// Mitsubishi GX Works2 project: ventilationUnitStart_exp   PLC: FX3G
// Базовая структура управления вентиляциооной установкой

// global labels: Global1
VAR_GLOBAL
  xStart AT M10 : BOOL;  (* Переменная разрешения на работу установки *)
  xSeason AT M12 : BOOL;  (* Определение сезона 0 - Зима 1 - Лето *)
  xAlarm AT M1 : BOOL;  (* Общий статус Аварий 0 - нет 1 - Авария *)
  xWarning AT M2 : BOOL;  (* Общий статус предупреждений 0 - нет 1 - есть предупреждения *)
  dI_AlarmFreeze AT X000 : BOOL;  (* Авария термостата заморозки *)
  xAlarmSensors AT M7 : BOOL;  (* Общая аврия Датчиков - всне диапазона *)
  dI_AlarmPumpWater AT X001 : BOOL;  (* Авария насоса (сработка защиты) *)
  dI_AlarmMotorSupply AT X002 : BOOL;  (* Авария реле Вентилятора Притока *)
  dI_AlarmMotorExhaust AT X003 : BOOL;  (* Авария реле Вентилятора Вытяжки *)
  dI_WarnPresFilterSupply AT X007 : BOOL;  (* Авария пресостата фильтра Притока *)
  dI_WarnPresFilterExaust AT X006 : BOOL;  (* Авария пресостата фильтра Вытяжки *)
  dI_AlarmPresMotorSupply AT X004 : BOOL;  (* Авария пресостата вентилятора Притока *)
  dI_AlarmPresMotorExhaust AT X005 : BOOL;  (* Авария пресостата вентилятора Вытяжки *)
  xAlarmWarmWater AT M8 : BOOL;  (* Авария снижения температуры теплоносителя темплообменника - Требуется прогрев *)
  wDeltaTempOut AT D11 : INT;  (* Значение смещения показаний датчика (корректировка) *)
  wDeltaTempInRoom AT D10 : INT;  (* Значение смещения показаний датчика (корректировка) *)
  wDeltaTempFromRoom AT D9 : INT;  (* Значение смещения показаний датчика (корректировка) *)
  wDeltaTempEmpty AT D8 : INT;  (* Значение смещения показаний датчика (корректировка) *)
  xAlarmSensorOut AT M6 : BOOL;  (* Авария датчика Наружней температуры *)
  xAlarmSensorInRoom AT M5 : BOOL;  (* Авария датчика температуры Подачи В помещение *)
  xAlarmSensorFromRoom AT M4 : BOOL;  (* Авария датчика температуры забираемого ИЗ помещения *)
  xAlarmSensorEmpty AT M3 : BOOL;  (* Авария датчика температуры *)
  iR_TempOut AT D6 : WORD;  (* Значение сопротивление линии связи резистивного датчика *)
  iR_TempInRoom AT D5 : WORD;  (* Значение сопротивление линии связи резистивного датчика *)
  iR_TempFromRoom AT D4 : WORD;  (* Значение сопротивление линии связи резистивного датчика *)
  iRTempEmpty AT D7 : WORD;  (* Значение сопротивление линии связи резистивного датчика *)
  dO_PumpStart AT Y004 : BOOL;  (* Разрешение на работу Насоса контура водяного теплообменника *)
  dO_SupplyMotorStart AT Y003 : BOOL;  (* Разрешение на запуск Вентилятора Притока *)
  dO_ExhaustMotorStart AT Y001 : BOOL;  (* Разрешение на запуск Вентилятора Вытяжки *)
  dO_SupplyDamperStart AT Y002 : BOOL;  (* Разрешение на открытие Заслонки Притока *)
  dO_ExhaustDamperStart AT Y000 : BOOL;  (* Разрешение на открытие Заслонки Вытяжки *)
  iDelayStart AT D2 : WORD;  (* Значение задержки (общее) *)
  iDelaySupplyMotor AT D3 : WORD;  (* Значение задержки пуска Вентилятора Притока *)
  iDelayExhaustMotor AT D1 : WORD;  (* Значение задержки пуска Вентилятора Вытяжки *)
  iDelayDamper AT D0 : WORD;  (* Значение задержки открытия заслонки *)
  xUserStart AT M11 : BOOL;  (* Переменная изменяемая Пользователем для разрешения работы *)
  xUserSeason AT M13 : BOOL;  (* Переменная изменяемая Пользователем для выбора Сезона *)
  xUserArarmReset AT M14 : BOOL;  (* Переменная изменяемая Пользователем для сброса общего флага Аварий *)
  xAlarmCritical AT M0 : BOOL;  (* Cтатус критических Аварий 0 - нет 1 - Авария *)
  xInit AT M15 : BOOL;  (* Переменная разрешающая иницилизацию при старте *)
  aI_TempOut AT D14 : INT;  (* AI_0 Датчик наружней температуры D8030 *)
  aI_TempSupply AT D15 : INT;  (* AI_1 Датчик притока (температуры подачи в помещение)  D8031 *)
  aI_TempWater AT D16 : INT;  (* AI_2 Датчик обратной воды  D8032 *)
  aI_TempRecupOut AT D17 : INT;  (* AI_3 Датчик температуры за рекуператором  D8033 *)
  aO_1 AT D8050 : REAL;  (* AO_ Первый аналоговый D8050 *)
  aO_2 AT D8051 : REAL;  (* AO_ Второй аналоговый выход D8051 *)
  iUserTempSummer AT D12 : INT;  (* Температура перехода на летний режим *)
  iUserTemWinter AT D13 : INT;  (* Температура перехода на зимний режим *)
  aI_TempFromRoom AT D18 : INT;  (* AI_4 Датчик вытяжной температуры из помещения D8034 *)
  iUserAccess AT D40 : WORD;  (* Уровень доступа текущего пользователя *)
  iUserSetpoint AT D20 : INT;  (* Уставка *)
  testTempOut AT D41 : INT;  (* Тестирование перехода   Зима/Лето *)
END_VAR

// task Task_01 (event TRUE, interval 0, priority 31): POU_01
// task Init (event TRUE, interval 0, priority 1): Init
// user libraries (not included): AlarmManger128, Utils

PROGRAM Init
VAR
  fbAmSet : AM_SET;
  fbAmInit : AM_INIT;
  fbAmIs : AM_HAS_ALARMS;
  fbAmBlockIs : AM_IS_BLOCK;
  fbAmEvents : AM_EVENT;
  fbAmRST : AM_RST;
  fbAmEventRST : AM_EVENT_RESET;
END_VAR
(*Programm is run only one time when plc started to initiate alarms,  warnings and configuration settings *)

(* Init PID*)

(*Init Alarms *)
IF NOT xInit THEN 
	AM_D_START :=3000; (* Start alarms library*)
	
	(* Critical Alarm signals*)
	 fbAmInit(iNum := 0, iSeverity :=4, iProcess :=1, xLock := TRUE, xLatch := TRUE,  xBuzzer := TRUE ); (*Fire alarm *)
	 fbAmInit(iNum := 1, iSeverity :=4, iProcess :=1, xLock := TRUE, xLatch := TRUE,  xBuzzer := TRUE ); (*Freeze alarm *)
	 fbAmInit(iNum := 2, iSeverity :=4, iProcess :=1, xLock := TRUE, xLatch := TRUE,  xBuzzer := TRUE ); (*Warming Up the water circuit*)
	 fbAmInit(iNum := 4, iSeverity :=4, iProcess :=1, xLock := TRUE, xLatch := TRUE,  xBuzzer := TRUE ); (*Critical alarm the water circuit*)
	  
	 (* Air Presure sensors*)
	 fbAmInit(iNum := 5, iSeverity :=2, iProcess :=2, xLock := TRUE, xLatch := FALSE,  xBuzzer := TRUE ); (*Supply filter *)
	 fbAmInit(iNum := 6, iSeverity :=2, iProcess :=2, xLock := TRUE, xLatch := FALSE,  xBuzzer := TRUE ); (*Exhaust filter *)
	 fbAmInit(iNum := 7, iSeverity :=3, iProcess :=2, xLock := TRUE, xLatch := FALSE,  xBuzzer := TRUE ); (*Supply motor air alarm *)
	 fbAmInit(iNum := 8, iSeverity :=3, iProcess :=2, xLock := TRUE, xLatch := FALSE,  xBuzzer := TRUE ); (*Exhaust motor air alarm *)
	 (* Vent Motors Alarm sensors*)
	 fbAmInit(iNum := 9, iSeverity :=3, iProcess :=3, xLock := TRUE, xLatch := FALSE,  xBuzzer := TRUE ); (*Supply motor Alarm *)
	 fbAmInit(iNum := 10, iSeverity :=3, iProcess :=3, xLock := TRUE, xLatch := FALSE,  xBuzzer := TRUE ); (*Exhaust motor Alarm *)
	 (* Pumpsr Alarm sensors*)
	 fbAmInit(iNum := 11, iSeverity :=3, iProcess :=3, xLock := TRUE, xLatch := FALSE,  xBuzzer := TRUE ); (*Pump water Alarm*)
	 fbAmInit(iNum := 12, iSeverity :=3, iProcess :=3, xLock := TRUE, xLatch := FALSE,  xBuzzer := TRUE ); (*Pump glycol Alarm*)
	 (* Temperature sensors*)
	 fbAmInit(iNum := 13, iSeverity :=2, iProcess :=4, xLock := TRUE, xLatch := FALSE,  xBuzzer := TRUE ); (*Temp out *)
	 fbAmInit(iNum := 14,  iSeverity :=2, iProcess :=4, xLock := TRUE, xLatch := FALSE,  xBuzzer := TRUE ); (*Temp supply in room *)
	 fbAmInit(iNum := 15,  iSeverity :=2, iProcess :=4, xLock := TRUE, xLatch := FALSE,  xBuzzer := TRUE ); (*Temp exhaust from room *)
	 fbAmInit(iNum := 16,  iSeverity :=2, iProcess :=4, xLock := TRUE, xLatch := FALSE,  xBuzzer := TRUE ); (*Temp after recuperation *)
	 fbAmInit(iNum := 17,  iSeverity :=2, iProcess :=4, xLock := TRUE, xLatch := FALSE,  xBuzzer := TRUE ); (*Temp water return *)
	 fbAmInit(iNum := 18,  iSeverity :=2, iProcess :=4, xLock := TRUE, xLatch := FALSE,  xBuzzer := TRUE ); (*Temp glycol return *)
	 
	 (* SeasonControl*)
	 fbAmInit(iNum := 30,  iSeverity :=1, iProcess :=5, xLock := FALSE, xLatch := FALSE,  xBuzzer := FALSE); (*start Winter Season *)
	 fbAmInit(iNum := 31,  iSeverity :=1, iProcess :=5, xLock := FALSE, xLatch := FALSE,  xBuzzer := FALSE); (*start SammerSeason *)
	 
	 (* Init ModBus*)
	 
	 
	 
	xInit := TRUE;	
END_IF ;

(* *)
END_PROGRAM

PROGRAM POU_01
VAR
  iStep : INT;
  fbAmSet : AM_SET;
  fbAmInit : AM_INIT;
  fbAmIs : AM_HAS_ALARMS;
  fbAmBlockIs : AM_IS_BLOCK;
  fbAmEvents : AM_EVENT;
  fbAmRST : AM_RST;
  fbAmEventRST : AM_EVENT_RESET;
  localSeasonTriger : BOOL;
  icountMin : INT;
  init : INT;
END_VAR
(* RST( MEP( xManualWorks ) , xAutoWorks );
RST( MEP(xAutoWorks ) ,xManualWorks  );  *)
(* System can work only in one state Auto or Manual There is constol change*)

(* IF iStep <> 10 THEN iStep := 0; END_IF; *)

CASE iStep OF
	0: (* Init *)
	IF xInit = 0  THEN 
		MOV(D14, 2, R23940); (* Инициализация входа AI01 (регистр R23940) как PT1000 - 2  *)
		MOV(D15, 2, R23941);
		MOV(D16, 2, R23942);
		MOV(D17, 2, R23943);
		xInit := 1;
	END_IF;
	iStep := 10;
	
	10: (* Base *)
	IF xUserStart = 1 THEN 
		iStep := 20;
		ELSE 
				xSeason := SeasonControl( aI_TempOut , iUserTemWinter , iUserTempSummer,  xUserSeason );
				IF MEP(xSeason) OR MEF(xSeason) THEN
					xUserSeason :=  xSeason ;
				END_IF;
		END_IF;
	20: (* Manage *)
		xSeason := 1;init
	END_CASE;



	
D500 := D100Z1;

IF MEP( M8013) AND xUserStart = TRUE  THEN
	icountMin := icountMin +1;
	IF icountMin =8 THEN
		icountMin := 0;

	END_IF;
END_IF;
END_PROGRAM

PROGRAM Process
VAR
  fbAmSet : AM_SET;
END_VAR
(*All proccess that works constantly - monit alarms, statuses and so on *)
(* Выполняем регистрацию события объявленного в программе Init при выполнении определенного (указываем при вызове) условия *)

(* Input  sensors Error - not data or conection from sensors conection*)
 (*iNum - number registred in Init programm Alarm  xState - condition for execution*)
fbAmSet(iNum:= 13, xState:= (D8030 = 32760) ); (*Temp out Error AI0 - D8030*)
fbAmSet(iNum:= 14, xState:= (D8031 = 32760) ); (*Temp supply in room Error AI1 - D8031*)
fbAmSet(iNum:= 15 ,xState:= (D8032 = 32760) ); (*Temp exhaust from room Error AI2 - D8032*)
fbAmSet(iNum:= 16 ,xState:= (D8033 = 32760) ); (*Temp after recuperation Error AI3 - D8033*)
fbAmSet(iNum:= 17 ,xState:= (D8034 = 32760) ); (*Temp water return Error AI4 - D8034*)
fbAmSet(iNum:= 18 ,xState:= (D8035 = 32760) ); (*Temp glycol return Error AI5 - D8035*)

(* Input values transmit to selected range*)
IF NOT (D8030 = 32760) THEN aI_TempOut := SCALE(D8030, 803,1, 1422,9, -500, 1100);ELSE aI_TempOut := 999; END_IF ;  
(*Проверяем входной порт D8030 на ошибку и сохраняем значение входа в переменную aI_TempOut если нет ошибки то с преобразованием входного значения в диапазоне от 803 до 1422 в выходной диапазон от 500 до 1100 Если ошибка есть назначаем - 999*)
IF NOT (D8031 = 32760) THEN aI_TempSupply:= SCALE(D8031, 803,1, 1422,9, -500, 1100);ELSE aI_TempSupply:= 999; END_IF ; (*aI_TempSupply *)
IF NOT (D8032 = 32760) THEN aI_TempWater := SCALE(D8032, 803,1, 1422,9, -500, 1100);ELSE aI_TempWater := 999; END_IF ;(*aI_TempWater *)
IF NOT (D8033 = 32760) THEN aI_TempRecupOut:= SCALE(D8033, 803,1, 1422,9, -500, 1100);ELSE aI_TempRecupOut:= 999; END_IF ;(*aI_TempRecupOut *)
	
(*Control of changes in the Season variable depending on the Outdoor Temperature *)
fbAmSet(iNum:= 30 ,xState:= (aI_TempOut > iUserTempSummer) );
fbAmSet(iNum:= 31 ,xState:= (aI_TempOut < iUserTemWinter) );
(* *)

(* *)

(* *)

(* *)
;
(* *)
END_PROGRAM

FUNCTION SeasonControl
VAR_INPUT
  tempOut : INT;  (* Temp Outdore - Температура наружнего воздуха *)
  tempWinter : INT;  (* Temp for switch on Winter - Уставка перехода на Зимний режим *)
  tempSummer : INT;  (* Temp for switch on Summer - Уставка перехода на летний режим *)
  triger : BOOL;  (* 1 - was switch to winter 0 - was switch to summer *)
END_VAR
	IF tempOut  <  tempWinter THEN 
		SeasonControl := 1; (* Output  Set flag - 1  to force switching to Winter *)
	ELSE 
		IF tempOut > tempSummer THEN 
			SeasonControl := 0; (* Output  Set flag - 0  to force switching to Summer*)
		ELSE 
			SeasonControl := triger; (* Don't change r*)
		END_IF;

	END_IF;
END_FUNCTION

FUNCTION TestFunction
TestFunction := TRUE;
END_FUNCTION
